{attribute 'GeneratedUsingTerminal: EL7201-0000-0017'}
{attribute addProperty BoxType "EL7201-0000-0017"}
{attribute addProperty Id "AdsAddrAT %I*AMSADDR8DcOutputShiftAT %I*DINT4DcInputShiftAT %I*DINT4Chn0AT %I*USINT1StateAT %I*UINT2"}
{attribute addProperty CRC "2529775534"}
{attribute addProperty Size "19"}
TYPE InfoData_96C94FAE EXTENDS InputBase_8311D824 :
STRUCT
	{attribute addProperty Name "AdsAddr"}
	AdsAddr AT %I* : AMSADDR;
	{attribute addProperty Name "DcOutputShift"}
	DcOutputShift AT %I* : DINT;
	{attribute addProperty Name "DcInputShift"}
	DcInputShift AT %I* : DINT;
	{attribute addProperty Name "Chn0"}
	Chn0 AT %I* : USINT;
	{attribute addProperty Name "State"}
	State AT %I* : UINT;
END_STRUCT
END_TYPE

(* stored: Version 1.2.0.0, ProductVersion 3.1.4024.11
   DUT InfoData_96C94FAE: Id {7cc5fd0b-cc07-44ca-8597-4113d44476af} *)
